FUNCTION_BLOCK CmdOneActuator (* CAT Function Block Type *)
  (* Standard: 61499-2 *)
  (* Version 0.0, 6/7/2026, Schneider Electric, template *)
  PACKAGE SE.Nereda;
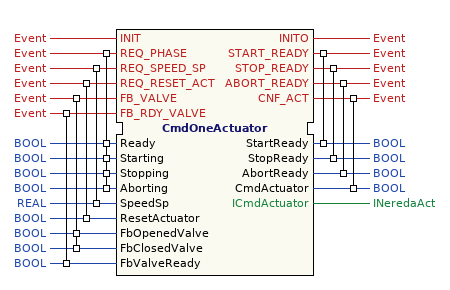
  EVENT_INPUT
    INIT;
    REQ_PHASE WITH Ready, Starting, Stopping, Aborting;
    REQ_SPEED_SP WITH SpeedSp;
    REQ_RESET_ACT WITH ResetActuator;
    FB_VALVE WITH FbOpenedValve, FbClosedValve;
    FB_RDY_VALVE WITH FbValveReady;
  END_EVENT
  EVENT_OUTPUT
    INITO;
    START_READY WITH StartReady;
    STOP_READY WITH StopReady;
    ABORT_READY WITH AbortReady;
    CNF_ACT WITH CmdActuator;
  END_EVENT
  VAR_INPUT
    Ready : BOOL;
    Starting : BOOL;
    Stopping : BOOL;
    Aborting : BOOL;
    SpeedSp : REAL;
    ResetActuator : BOOL;
    FbOpenedValve : BOOL;
    FbClosedValve : BOOL;
    FbValveReady : BOOL;
  END_VAR
  VAR_OUTPUT
    StartReady : BOOL;
    StopReady : BOOL;
    AbortReady : BOOL;
    CmdActuator : BOOL;
  END_VAR
  PLUGS
    ICmdActuator : INeredaAct;
  END_PLUGS
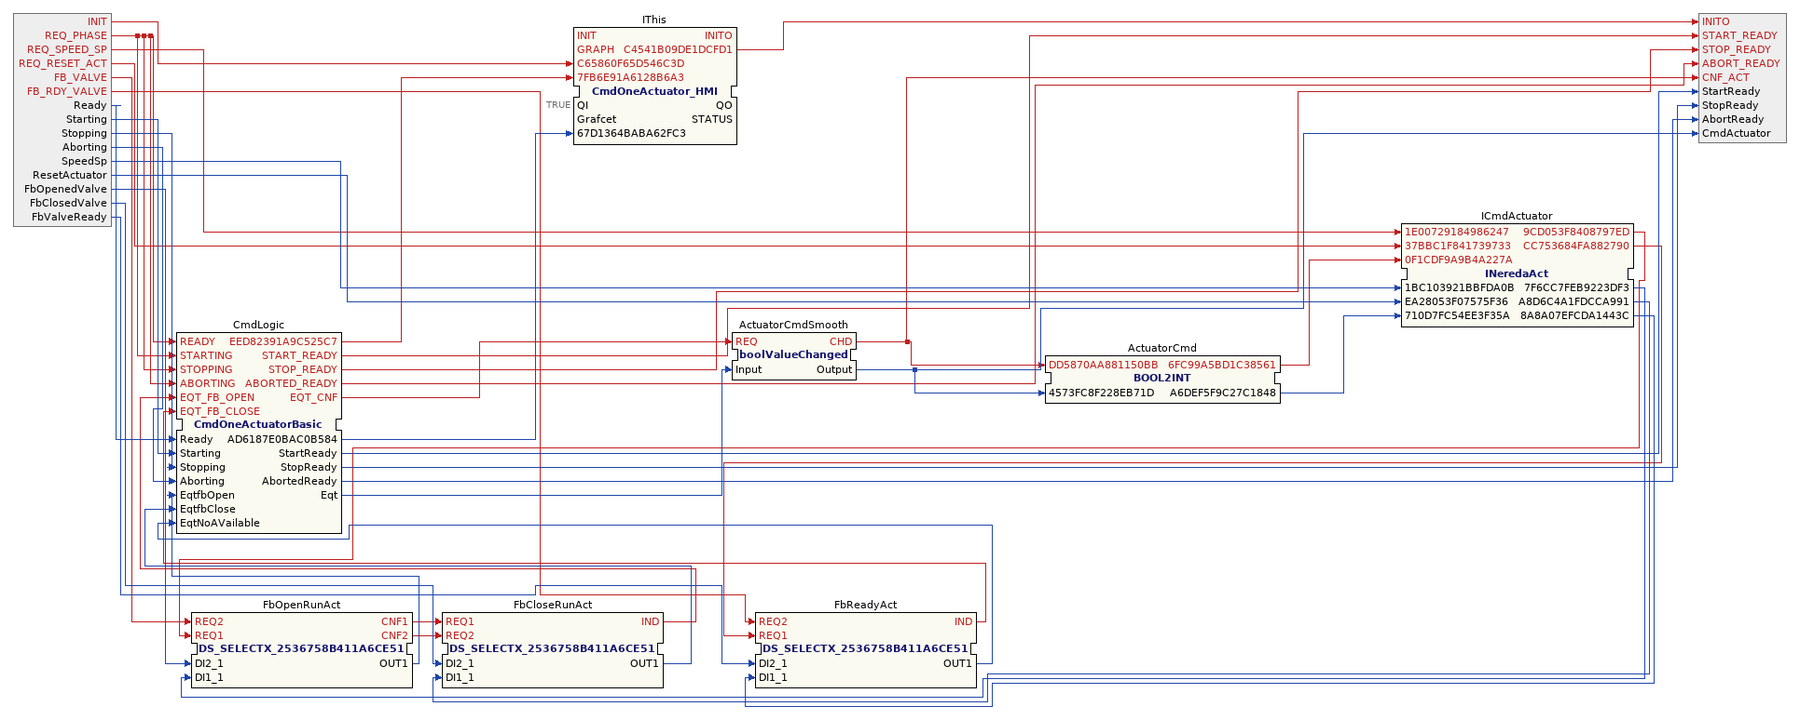
  (* 01 - FUNCTIONNAL INPUT INTERFACE *)
  (* 00 - INITIALIZATION *)
  (* 05 - LOGIC *)
  (* 06 - HMI INTERFACE *)
  (* 03 - FIELD INTERFACE *)
  (* 02 - FUNCTIONNAL OUTPUT INTERFACE *)
  (* Command Logic *)
  FBS
    IThis : CmdOneActuator_HMI(QI := TRUE);
    ActuatorCmdSmooth : boolValueChanged;
    FbOpenRunAct : DS_SELECTX_2536758B411A6CE51; {SET_ATTRIBUTE(Configuration.GenericFBType.InterfaceParams, Runtime.Standard#CNTX:=2;CNTY:=1;DI${CNTX,_,CNTY$}:BOOL)}
    FbCloseRunAct : DS_SELECTX_2536758B411A6CE51; {SET_ATTRIBUTE(Configuration.GenericFBType.InterfaceParams, Runtime.Standard#CNTX:=2;CNTY:=1;DI${CNTX,_,CNTY$}:BOOL)}
    FbReadyAct : DS_SELECTX_2536758B411A6CE51; {SET_ATTRIBUTE(Configuration.GenericFBType.InterfaceParams, Runtime.Standard#CNTX:=2;CNTY:=1;DI${CNTX,_,CNTY$}:BOOL)}
    CmdLogic : CmdOneActuatorBasic;
    ActuatorCmd : BOOL2INT;
  END_FBS
  EVENT_CONNECTIONS
    ActuatorCmdSmooth.CHD TO CNF_ACT;
    FB_VALVE TO FbOpenRunAct.REQ2;
    FbOpenRunAct.CNF1 TO FbCloseRunAct.REQ1;
    FbOpenRunAct.CNF2 TO FbCloseRunAct.REQ2;
    FB_RDY_VALVE TO FbReadyAct.REQ2;
    INIT TO IThis.C65860F65D546C3D;
    IThis.C4541B09DE1DCFD1 TO INITO;
    CmdLogic.EED82391A9C525C7 TO IThis.7FB6E91A6128B6A3;
    REQ_PHASE TO CmdLogic.READY;
    REQ_PHASE TO CmdLogic.STARTING;
    REQ_PHASE TO CmdLogic.STOPPING;
    REQ_PHASE TO CmdLogic.ABORTING;
    REQ_SPEED_SP TO ICmdActuator.1E00729184986247;
    REQ_RESET_ACT TO ICmdActuator.37BBC1F841739733;
    CmdLogic.START_READY TO START_READY;
    CmdLogic.STOP_READY TO STOP_READY;
    CmdLogic.ABORTED_READY TO ABORT_READY;
    ActuatorCmdSmooth.CHD TO ActuatorCmd.DD5870AA881150BB;
    ActuatorCmd.6FC99A5BD1C38561 TO ICmdActuator.0F1CDF9A9B4A227A;
    CmdLogic.EQT_CNF TO ActuatorCmdSmooth.REQ;
    ICmdActuator.9CD053F8408797ED TO FbOpenRunAct.REQ1;
    ICmdActuator.CC753684FA882790 TO FbReadyAct.REQ1;
    FbCloseRunAct.IND TO CmdLogic.EQT_FB_OPEN;
    FbReadyAct.IND TO CmdLogic.EQT_FB_CLOSE;
  END_CONNECTIONS
  DATA_CONNECTIONS
    ActuatorCmdSmooth.Output TO CmdActuator;
    FbOpenedValve TO FbOpenRunAct.DI2_1;
    FbClosedValve TO FbCloseRunAct.DI2_1;
    FbValveReady TO FbReadyAct.DI2_1;
    CmdLogic.AD6187E0BAC0B584 TO IThis.67D1364BABA62FC3;
    Ready TO CmdLogic.Ready;
    Starting TO CmdLogic.Starting;
    Stopping TO CmdLogic.Stopping;
    Aborting TO CmdLogic.Aborting;
    SpeedSp TO ICmdActuator.1BC103921BBFDA0B;
    ResetActuator TO ICmdActuator.EA28053F07575F36;
    CmdLogic.StartReady TO StartReady;
    CmdLogic.StopReady TO StopReady;
    CmdLogic.AbortedReady TO AbortReady;
    ActuatorCmdSmooth.Output TO ActuatorCmd.4573FC8F228EB71D;
    ActuatorCmd.A6DEF5F9C27C1848 TO ICmdActuator.710D7FC54EE3F35A;
    CmdLogic.Eqt TO ActuatorCmdSmooth.Input;
    ICmdActuator.7F6CC7FEB9223DF3 TO FbOpenRunAct.DI1_1;
    ICmdActuator.A8D6C4A1FDCCA991 TO FbCloseRunAct.DI1_1;
    ICmdActuator.8A8A07EFCDA1443C TO FbReadyAct.DI1_1;
    FbOpenRunAct.OUT1 TO CmdLogic.EqtfbOpen;
    FbCloseRunAct.OUT1 TO CmdLogic.EqtfbClose;
    FbReadyAct.OUT1 TO CmdLogic.EqtNoAVailable;
  END_CONNECTIONS
END_FUNCTION_BLOCK
